TYPE ST_System_AFA_Zustand :
STRUCT
	Betrieb_Anford			: BOOL;
	Betrieb_Soll				: BOOL;
	Betrieb					: BOOL;

	Regelung_Modus			: SINT;
	Regelung_Sollw			: REAL;
	Regelung_Sollw_Anford	: REAL;
	Regelung_Stellw			: REAL;

	Modus_Waermeabsorption				: BOOL;
	Modus_Rueckkuehlung				: BOOL;
	Modus_Netz			: BOOL;
	Modus_viaWanddeckentemperierung	: BOOL;

	Temp_Aussen			: REAL;
	Temp_Fassade_Ost		: REAL;
	Temp_Fassade_West		: REAL;
	Temp_Fassade_Decke	: REAL;
	Temp_stellbar_Max		: REAL;
	Temp_stellbar_Min		: REAL;
	Temp_Rueckl_Ost		: REAL;
	Temp_Rueckl_West		: REAL;
	Temp_Ruecklauf		: REAL;

	Kommunikation			: BOOL	:= FALSE;	(* Kommunikation zu IWB Bauteil Monitoring *)


	Systemdruck				: REAL;

	Freigabe					: BOOL;
	Freigabe_Deakt			: BOOL;
	Freigabe_Code			: WORD;

	Stoerung					: BOOL;
	Stoerung_Code			: WORD;

	Warnung					: BOOL;
	Warnung_Code			: WORD;

	Status					: SINT;
	Status_Vorl_Pumpen		: BOOL;
	Status_Vorl_Regelventil	: BOOL;
	Status_Nachl_Pumpen		: BOOL;
	Status_Nachl_Regelventil	: BOOL;
	Status_Wiedereinschalten	: BOOL;

	Quittierung				: BOOL;

END_STRUCT
END_TYPE

(* stored: Version 1.1.0.1, ProductVersion 3.1.4024.9
   DUT ST_System_AFA_Zustand: Id {706e94a4-666f-44cc-942f-773a54eb5592} *)
